// SIMATIC STEP 7 (V5.x) project S7_m1
// CPU: CPU312(1)
// station: P_ADR_BUS
// station: Hardware
// station: SIMATIC 300 Station
// program: S7 Program(1)

SYMBOL_TABLE
"start"	I 0.0	BOOL
"stop"	I 0.1	BOOL
"green2"	Q 0.0	BOOL
"yellow2"	Q 0.1	BOOL
"red2"	Q 0.2	BOOL
"green1"	Q 0.3	BOOL
"yellow1"	Q 0.4	BOOL
"red1"	Q 0.5	BOOL
"start(light)"	Q 0.6	BOOL
"stop(light)"	Q 0.7	BOOL
END_SYMBOL_TABLE

ORGANIZATION_BLOCK OB 1
TITLE = "Main Program Sweep (Cycle)"
VERSION : 0.1
VAR_TEMP
  OB1_EV_CLASS : BYTE ;	//Bits 0-3 = 1 (Coming event), Bits 4-7 = 1 (Event class 1)
  OB1_SCAN_1 : BYTE ;	//1 (Cold restart scan 1 of OB 1), 3 (Scan 2-n of OB 1)
  OB1_PRIORITY : BYTE ;	//Priority of OB Execution
  OB1_OB_NUMBR : BYTE ;	//1 (Organization block 1, OB1)
  OB1_RESERVED_1 : BYTE ;	//Reserved for system
  OB1_RESERVED_2 : BYTE ;	//Reserved for system
  OB1_PREV_CYCLE : INT ;	//Cycle time of previous OB1 scan (milliseconds)
  OB1_MIN_CYCLE : INT ;	//Minimum cycle time of OB1 (milliseconds)
  OB1_MAX_CYCLE : INT ;	//Maximum cycle time of OB1 (milliseconds)
  OB1_DATE_TIME : DATE_AND_TIME ;	//Date and time OB1 started
END_VAR
BEGIN
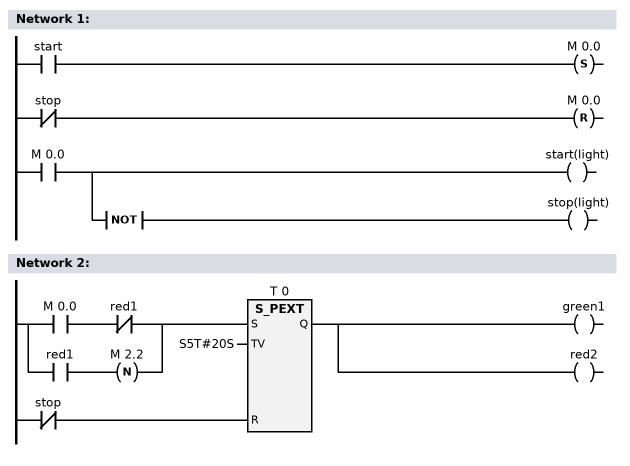
NETWORK
TITLE =
      A     "start";
      S     M 0.0;
      AN    "stop";
      R     M 0.0;
      A     M 0.0;
      =     L 20.0;
      A     L 20.0;
      BLD   102;
      =     "start(light)";
      A     L 20.0;
      NOT;
      =     "stop(light)";
NETWORK
TITLE =
      A(;
      A     M 0.0;
      AN    "red1";
      O(;
      A     "red1";
      FN    M 2.2;
      );
      );
      L     S5T#20S;
      SE    T 0;
      AN    "stop";
      R     T 0;
      NOP   0;
      NOP   0;
      A     T 0;
      =     "green1";
      =     "red2";
NETWORK
TITLE =
      A(;
      A     M 0.0;
      A     "green1";
      FN    M 1.1;
      S     M 1.0;
      A(;
      ON    "stop";
      O     T 0;
      );
      R     M 1.0;
      A     M 1.0;
      );
      L     S5T#7S;
      SE    T 1;
      AN    "stop";
      R     T 1;
      NOP   0;
      NOP   0;
      A     T 1;
      =     "yellow1";
      =     "yellow2";
NETWORK
TITLE =
      A(;
      A     M 0.0;
      A     "yellow1";
      FN    M 2.1;
      S     M 2.0;
      A(;
      ON    "stop";
      O     T 1;
      );
      R     M 2.0;
      A     M 2.0;
      );
      L     S5T#20S;
      SE    T 2;
      AN    "stop";
      R     T 2;
      NOP   0;
      NOP   0;
      A     T 2;
      =     "red1";
      =     "green2";
END_ORGANIZATION_BLOCK
